{attribute addProperty BoxType "EK1100-0000-0018"}
{attribute addProperty Id "Beckhoff_EL7xxxEK1122Beckhoff_EL7xxxEK1122_D459DE4F162A_0001_EL7031_0000_0016EL7031_F0B8B72B21827.25A_0002_EL7031_0000_0017EL7031_F0B8B72B21827.25A_0003_EL7031_0000_0018EL7031_D3B817C722628.25A_0004_EL7031_0000_0019EL7031_D3B817C722628.25A_0005_EL7031_0000_0020EL7031_D3B817C722628.25A_0006_EL7031_0000_0021EL7031_D3B817C722628.25A_0007_EL7031_0000_0022EL7031_D3B817C722628.25A_0008_EL7031_0000_0023EL7031_26D8313822628.25A_0009_EL7031_0000_0024EL7031_26D8313822628.25A_0010_EL7031_0000_0025EL7031_26D8313822628.25A_0011_EL7031_0000_0026EL7031_26D8313822628.25A_0012_EL7031_0030_0016EL7031_FC4B957935444.25A_0013_EL7037_0000_0016EL7037_F30AD12822628.25A_0014_EL7037_0000_0017EL7037_F30AD12822628.25A_0015_EL7037_0000_0018EL7037_F30AD12822628.25A_0016_EL7037_0000_0019EL7037_F30AD12822628.25A_0017_EL7037_0000_0020EL7037_F30AD12822628.25A_0018_EL7041_0000_0016EL7041_F90A638921827.25A_0019_EL7041_0000_0017EL7041_F90A638921827.25A_0020_EL7041_0000_0018EL7041_DA0AC36522628.25A_0021_EL7041_0000_0019EL7041_DA0AC36522628.25A_0022_EL7041_0000_0020EL7041_DA0AC36522628.25A_0023_EL7041_0000_0021EL7041_DA0AC36522628.25A_0024_EL7041_0000_0022EL7041_DA0AC36522628.25A_0025_EL7041_0000_0023EL7041_992C246822628.25A_0026_EL7041_0000_0024EL7041_992C246822628.25A_0027_EL7041_0000_0025EL7041_992C246822628.25A_0028_EL7041_0001_0016EL7041_086BBB4B24630.75A_0029_EL7041_0001_0017EL7041_DC8AD8ED21827.25A_0030_EL7041_0001_0018EL7041_FF8A780122628.25A_0031_EL7041_0001_0019EL7041_FF8A780122628.25A_0032_EL7041_0001_0020EL7041_FF8A780122628.25A_0033_EL7041_0001_0021EL7041_FF8A780122628.25A_0034_EL7041_0001_0022EL7041_4E04BDA322628.25A_0035_EL7041_0001_0023EL7041_4E04BDA322628.25A_0036_EL7041_0001_0024EL7041_4E04BDA322628.25A_0037_EL7041_0052_0016EL7041_26D8313822628.25A_0038_EL7041_1000_0016EL7041_F90A638921827.25A_0039_EL7041_1000_0017EL7041_F90A638921827.25A_0040_EL7041_1000_0018EL7041_F90A638921827.25A_0041_EL7041_1000_0019EL7041_F90A638921827.25A_0042_EL7041_1000_0020EL7041_BA2C848421827.25A_0043_EL7041_1000_0021EL7041_BA2C848421827.25A_0044_EL7047_0000_0016EL7047_F30AD12822628.25A_0045_EL7047_0000_0017EL7047_F30AD12822628.25A_0046_EL7047_0000_0018EL7047_F30AD12822628.25A_0047_EL7047_0000_0019EL7047_F30AD12822628.25A_0048_EL7047_0000_0020EL7047_F30AD12822628.25A_0049_EL7047_0000_0021EL7047_F30AD12822628.25A_0050_EL7047_9014_0021EL7047_F30AD12822628.25A_0051_EL7411_0000_0016EL7411_675FBD0529036.25A_0052_EL7411_0000_0017EL7411_675FBD0529036.25A_0053_EL7411_0000_0018EL7411_675FBD0529036.25"}
{attribute addProperty CRC "2435900283"}
{attribute addProperty SizeInBites "12246"}
{attribute addProperty SizeInBytes "1530.75"}
TYPE Beckhoff_EL7xxx_9130E37B EXTENDS EK1100_179A0949 :
STRUCT
	{attribute addProperty Name "Beckhoff_EL7xxxEK1122"}
	Beckhoff_EL7xxxEK1122 : Beckhoff_EL7xxxEK1122_D459DE4F;
	{attribute addProperty Name "A_0001_EL7031_0000_0016"}
	A_0001_EL7031_0000_0016 : EL7031_F0B8B72B;
	{attribute addProperty Name "A_0002_EL7031_0000_0017"}
	A_0002_EL7031_0000_0017 : EL7031_F0B8B72B;
	{attribute addProperty Name "A_0003_EL7031_0000_0018"}
	A_0003_EL7031_0000_0018 : EL7031_D3B817C7;
	{attribute addProperty Name "A_0004_EL7031_0000_0019"}
	A_0004_EL7031_0000_0019 : EL7031_D3B817C7;
	{attribute addProperty Name "A_0005_EL7031_0000_0020"}
	A_0005_EL7031_0000_0020 : EL7031_D3B817C7;
	{attribute addProperty Name "A_0006_EL7031_0000_0021"}
	A_0006_EL7031_0000_0021 : EL7031_D3B817C7;
	{attribute addProperty Name "A_0007_EL7031_0000_0022"}
	A_0007_EL7031_0000_0022 : EL7031_D3B817C7;
	{attribute addProperty Name "A_0008_EL7031_0000_0023"}
	A_0008_EL7031_0000_0023 : EL7031_26D83138;
	{attribute addProperty Name "A_0009_EL7031_0000_0024"}
	A_0009_EL7031_0000_0024 : EL7031_26D83138;
	{attribute addProperty Name "A_0010_EL7031_0000_0025"}
	A_0010_EL7031_0000_0025 : EL7031_26D83138;
	{attribute addProperty Name "A_0011_EL7031_0000_0026"}
	A_0011_EL7031_0000_0026 : EL7031_26D83138;
	{attribute addProperty Name "A_0012_EL7031_0030_0016"}
	A_0012_EL7031_0030_0016 : EL7031_FC4B9579;
	{attribute addProperty Name "A_0013_EL7037_0000_0016"}
	A_0013_EL7037_0000_0016 : EL7037_F30AD128;
	{attribute addProperty Name "A_0014_EL7037_0000_0017"}
	A_0014_EL7037_0000_0017 : EL7037_F30AD128;
	{attribute addProperty Name "A_0015_EL7037_0000_0018"}
	A_0015_EL7037_0000_0018 : EL7037_F30AD128;
	{attribute addProperty Name "A_0016_EL7037_0000_0019"}
	A_0016_EL7037_0000_0019 : EL7037_F30AD128;
	{attribute addProperty Name "A_0017_EL7037_0000_0020"}
	A_0017_EL7037_0000_0020 : EL7037_F30AD128;
	{attribute addProperty Name "A_0018_EL7041_0000_0016"}
	A_0018_EL7041_0000_0016 : EL7041_F90A6389;
	{attribute addProperty Name "A_0019_EL7041_0000_0017"}
	A_0019_EL7041_0000_0017 : EL7041_F90A6389;
	{attribute addProperty Name "A_0020_EL7041_0000_0018"}
	A_0020_EL7041_0000_0018 : EL7041_DA0AC365;
	{attribute addProperty Name "A_0021_EL7041_0000_0019"}
	A_0021_EL7041_0000_0019 : EL7041_DA0AC365;
	{attribute addProperty Name "A_0022_EL7041_0000_0020"}
	A_0022_EL7041_0000_0020 : EL7041_DA0AC365;
	{attribute addProperty Name "A_0023_EL7041_0000_0021"}
	A_0023_EL7041_0000_0021 : EL7041_DA0AC365;
	{attribute addProperty Name "A_0024_EL7041_0000_0022"}
	A_0024_EL7041_0000_0022 : EL7041_DA0AC365;
	{attribute addProperty Name "A_0025_EL7041_0000_0023"}
	A_0025_EL7041_0000_0023 : EL7041_992C2468;
	{attribute addProperty Name "A_0026_EL7041_0000_0024"}
	A_0026_EL7041_0000_0024 : EL7041_992C2468;
	{attribute addProperty Name "A_0027_EL7041_0000_0025"}
	A_0027_EL7041_0000_0025 : EL7041_992C2468;
	{attribute addProperty Name "A_0028_EL7041_0001_0016"}
	A_0028_EL7041_0001_0016 : EL7041_086BBB4B;
	{attribute addProperty Name "A_0029_EL7041_0001_0017"}
	A_0029_EL7041_0001_0017 : EL7041_DC8AD8ED;
	{attribute addProperty Name "A_0030_EL7041_0001_0018"}
	A_0030_EL7041_0001_0018 : EL7041_FF8A7801;
	{attribute addProperty Name "A_0031_EL7041_0001_0019"}
	A_0031_EL7041_0001_0019 : EL7041_FF8A7801;
	{attribute addProperty Name "A_0032_EL7041_0001_0020"}
	A_0032_EL7041_0001_0020 : EL7041_FF8A7801;
	{attribute addProperty Name "A_0033_EL7041_0001_0021"}
	A_0033_EL7041_0001_0021 : EL7041_FF8A7801;
	{attribute addProperty Name "A_0034_EL7041_0001_0022"}
	A_0034_EL7041_0001_0022 : EL7041_4E04BDA3;
	{attribute addProperty Name "A_0035_EL7041_0001_0023"}
	A_0035_EL7041_0001_0023 : EL7041_4E04BDA3;
	{attribute addProperty Name "A_0036_EL7041_0001_0024"}
	A_0036_EL7041_0001_0024 : EL7041_4E04BDA3;
	{attribute addProperty Name "A_0037_EL7041_0052_0016"}
	A_0037_EL7041_0052_0016 : EL7041_26D83138;
	{attribute addProperty Name "A_0038_EL7041_1000_0016"}
	A_0038_EL7041_1000_0016 : EL7041_F90A6389;
	{attribute addProperty Name "A_0039_EL7041_1000_0017"}
	A_0039_EL7041_1000_0017 : EL7041_F90A6389;
	{attribute addProperty Name "A_0040_EL7041_1000_0018"}
	A_0040_EL7041_1000_0018 : EL7041_F90A6389;
	{attribute addProperty Name "A_0041_EL7041_1000_0019"}
	A_0041_EL7041_1000_0019 : EL7041_F90A6389;
	{attribute addProperty Name "A_0042_EL7041_1000_0020"}
	A_0042_EL7041_1000_0020 : EL7041_BA2C8484;
	{attribute addProperty Name "A_0043_EL7041_1000_0021"}
	A_0043_EL7041_1000_0021 : EL7041_BA2C8484;
	{attribute addProperty Name "A_0044_EL7047_0000_0016"}
	A_0044_EL7047_0000_0016 : EL7047_F30AD128;
	{attribute addProperty Name "A_0045_EL7047_0000_0017"}
	A_0045_EL7047_0000_0017 : EL7047_F30AD128;
	{attribute addProperty Name "A_0046_EL7047_0000_0018"}
	A_0046_EL7047_0000_0018 : EL7047_F30AD128;
	{attribute addProperty Name "A_0047_EL7047_0000_0019"}
	A_0047_EL7047_0000_0019 : EL7047_F30AD128;
	{attribute addProperty Name "A_0048_EL7047_0000_0020"}
	A_0048_EL7047_0000_0020 : EL7047_F30AD128;
	{attribute addProperty Name "A_0049_EL7047_0000_0021"}
	A_0049_EL7047_0000_0021 : EL7047_F30AD128;
	{attribute addProperty Name "A_0050_EL7047_9014_0021"}
	A_0050_EL7047_9014_0021 : EL7047_F30AD128;
	{attribute addProperty Name "A_0051_EL7411_0000_0016"}
	A_0051_EL7411_0000_0016 : EL7411_675FBD05;
	{attribute addProperty Name "A_0052_EL7411_0000_0017"}
	A_0052_EL7411_0000_0017 : EL7411_675FBD05;
	{attribute addProperty Name "A_0053_EL7411_0000_0018"}
	A_0053_EL7411_0000_0018 : EL7411_675FBD05;
END_STRUCT
END_TYPE

(* stored: Version 1.2.0.0, ProductVersion 3.1.4024.9
   DUT Beckhoff_EL7xxx_9130E37B: Id {884a6ae3-507a-4e32-a10c-7e69a3933ebb} *)
